(*

.. <legal notes>

legal notes
=================
| SPDX-FileCopyrightText: © 2026 Oleksandr Tiutyk <trofimich@gmail.com>
| SPDX-License-Identifier: LGPL-3.0-only
| For details check: LGPL-3.0-only_

.. _LGPL-3.0-only: https://www.gnu.org/licenses/lgpl-3.0.en.html

.. </legal notes>

*)

INTERFACE ISimulatable EXTENDS Core.IObject

{attribute 'monitoring' := 'call'}
PROPERTY SimulationMode : BOOL
GET
END_GET
END_PROPERTY

END_INTERFACE

(* stored: Version 1.1.0.1
   Itf ISimulatable: Id {64def839-9c7f-49fb-bb6c-6e139237e3fc}
   Property SimulationMode: Id {f5dfb847-33cc-4380-a1cf-0d2edbb1a6ef}
   Get Get: Id {26bbacea-8cbd-4c03-a1df-2721a1043836} *)
